(* CODESYS project proyectoFinal.project

Project tree, tasks and I/O mapping:
  Device : CODESYS Control Win V3, 3S - Smart Software Solutions GmbH, version 3.5.12.60
    application Application
      libraries: Standard, * (System)
      task MainTask (cyclic, interval t#20ms, priority 1) calls PLC_PRG
      task VISU_TASK (cyclic, interval 100 ms, priority 31) calls VisuElems.Visu_Prg
      program PLC_PRG [LD]
      visualisation Visualization
      function block LEVELMETER [LD]
      function block LEVEL_SENSORS [LD]
      function block TANK_CONTROLER [LD]
      function block LIGHTHING [LD]
      function block TIMER [LD]
      function block STATES_MACHINE [LD]
      function block TEMPERATURE_ANALOG [LD]
      function block ANALOG_TEMPERATURE [LD]
      function block TEMPERATURE_CONTROLER [LD]
      program HEATING [LD]
  text list GlobalTextList
*)

// Device/Application/PLC_PRG
	PROGRAM PLC_PRG
VAR RETAIN
	start: BOOL;
	t: TIME;
	sweet_selected: BOOL;
	acid_selected: BOOL;
	bitter_selected: BOOL;
	state_filling_mixture: BOOL;
	state_filling_solids: BOOL;
	state_sweet: BOOL;
	state_acid: BOOL;
	state_bitter: BOOL;
	state_ending: BOOL;
	state_emptying: BOOL;
	state_emergency: BOOL;
	count:BOOL;
	level: REAL;
	state_ready: BOOL;
END_VAR
VAR
	emergency_lamp: BOOL;
	speed: REAL;
	sensor_lvl_110: BOOL;
	sensed_level: REAL;
	start_button: BOOL;
	sweet_button: BOOL;
	acid_button: BOOL;
	bitter_button: BOOL;
	stop_button: BOOL;
	sensor_lvl_0: BOOL;
	sensor_lvl_60: BOOL;
	sensor_lvl_100: BOOL;
	empty_button: BOOL;
	filling_mixture_lamp: BOOL;
	filling_solids_lamp: BOOL;
	in_process_lamp: BOOL;
	sweet_selected_lamp: BOOL;
	acid_selected_lamp: BOOL;
	bitter_selected_lamp: BOOL;
	ending_lamp: BOOL;
	emptying_lamp: BOOL;
	ready_lamp: BOOL;
	reset: BOOL;
	TIMER_0: TIMER;
	STATES_MACHINE_0: STATES_MACHINE;
	LEVELMETER_0: LEVELMETER;
	LEVEL_SENSORS_0: LEVEL_SENSORS;
	TANK_CONTROLER_0: TANK_CONTROLER;
	mixer_lamp: BOOL;
	mixture_valve: BOOL;
	solids_band: BOOL;
	LIGHTHING_0: LIGHTHING;
	lighthing_lamp: BOOL;
	color: DWORD;
	wave_length: INT;
	TEMPERATURE_METER_0: TEMPERATURE_ANALOG;
	sensor_analog: REAL;
	temp: REAL:=20;
	ANALOG_TEMPERATURE_0: ANALOG_TEMPERATURE;
	sensed_temperature: REAL;
	TEMP_CONTROLER_0: TEMPERATURE_CONTROLER;
	heat: BOOL;
	empty_valve: INT;
	empty_valve_lamp: BOOL;
END_VAR
VAR // added by the converter: edge detectors and wires of the graphical bodies
    _w1 : BOOL;
END_VAR

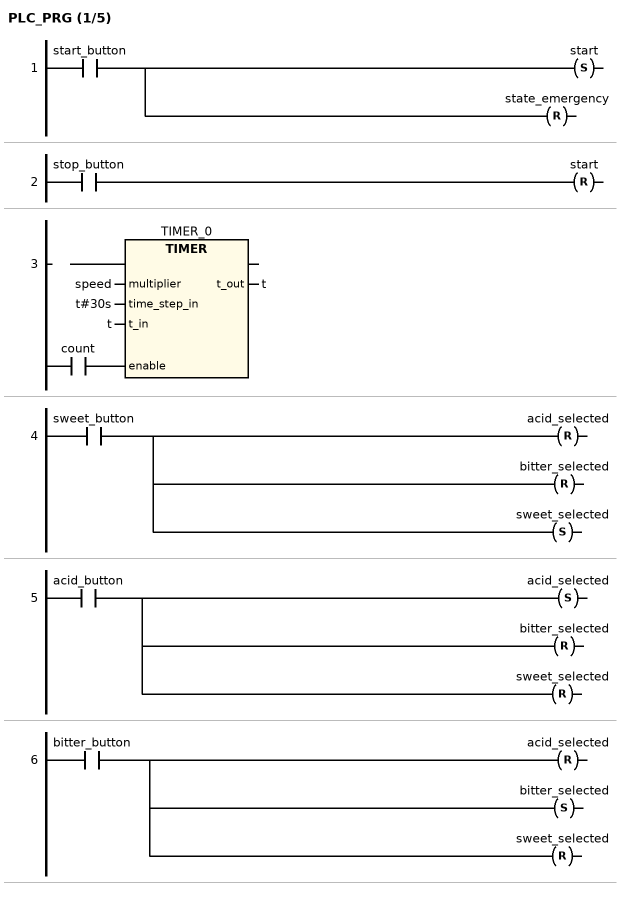
// NETWORK 1
start S= start_button;
state_emergency R= start_button;

// NETWORK 2
start R= stop_button;

// NETWORK 3
TIMER_0(multiplier := speed, time_step_in := t#30s, t_in := t, enable := count, t_out => t); // TIMER

// NETWORK 4
acid_selected R= sweet_button;
bitter_selected R= sweet_button;
sweet_selected S= sweet_button;

// NETWORK 5
acid_selected S= acid_button;
bitter_selected R= acid_button;
sweet_selected R= acid_button;

// NETWORK 6
acid_selected R= bitter_button;
bitter_selected S= bitter_button;
sweet_selected R= bitter_button;

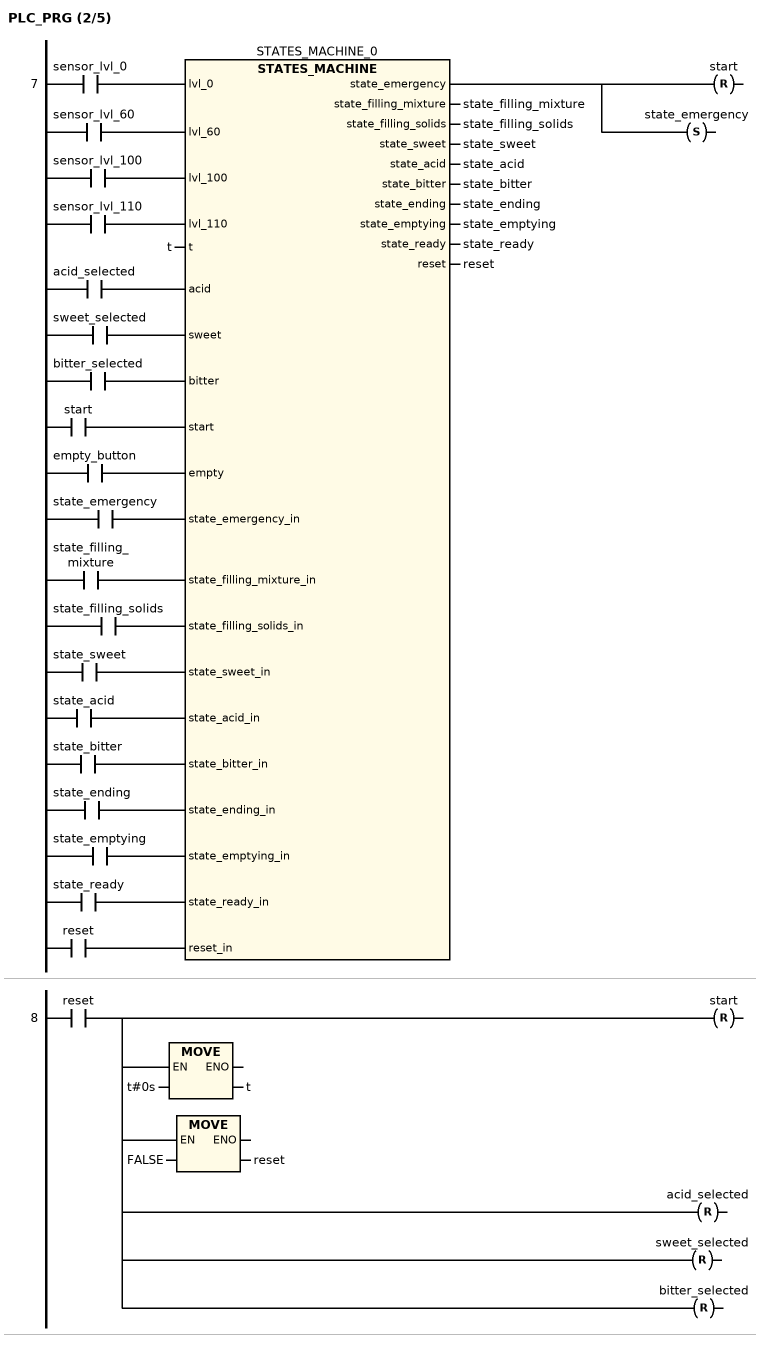
// NETWORK 7
STATES_MACHINE_0(
    lvl_0 := sensor_lvl_0,
    lvl_60 := sensor_lvl_60,
    lvl_100 := sensor_lvl_100,
    lvl_110 := sensor_lvl_110,
    t := t,
    acid := acid_selected,
    sweet := sweet_selected,
    bitter := bitter_selected,
    start := start,
    empty := empty_button,
    state_emergency_in := state_emergency,
    state_filling_mixture_in := state_filling_mixture,
    state_filling_solids_in := state_filling_solids,
    state_sweet_in := state_sweet,
    state_acid_in := state_acid,
    state_bitter_in := state_bitter,
    state_ending_in := state_ending,
    state_emptying_in := state_emptying,
    state_ready_in := state_ready,
    reset_in := reset,
    state_filling_mixture => state_filling_mixture,
    state_filling_solids => state_filling_solids,
    state_sweet => state_sweet,
    state_acid => state_acid,
    state_bitter => state_bitter,
    state_ending => state_ending,
    state_emptying => state_emptying,
    state_ready => state_ready,
    reset => reset); // STATES_MACHINE
start R= STATES_MACHINE_0.state_emergency;
state_emergency S= STATES_MACHINE_0.state_emergency;

// NETWORK 8
_w1 := reset;
start R= _w1;
IF _w1 THEN t := t#0s; END_IF
IF _w1 THEN reset := FALSE; END_IF
acid_selected R= _w1;
sweet_selected R= _w1;
bitter_selected R= _w1;

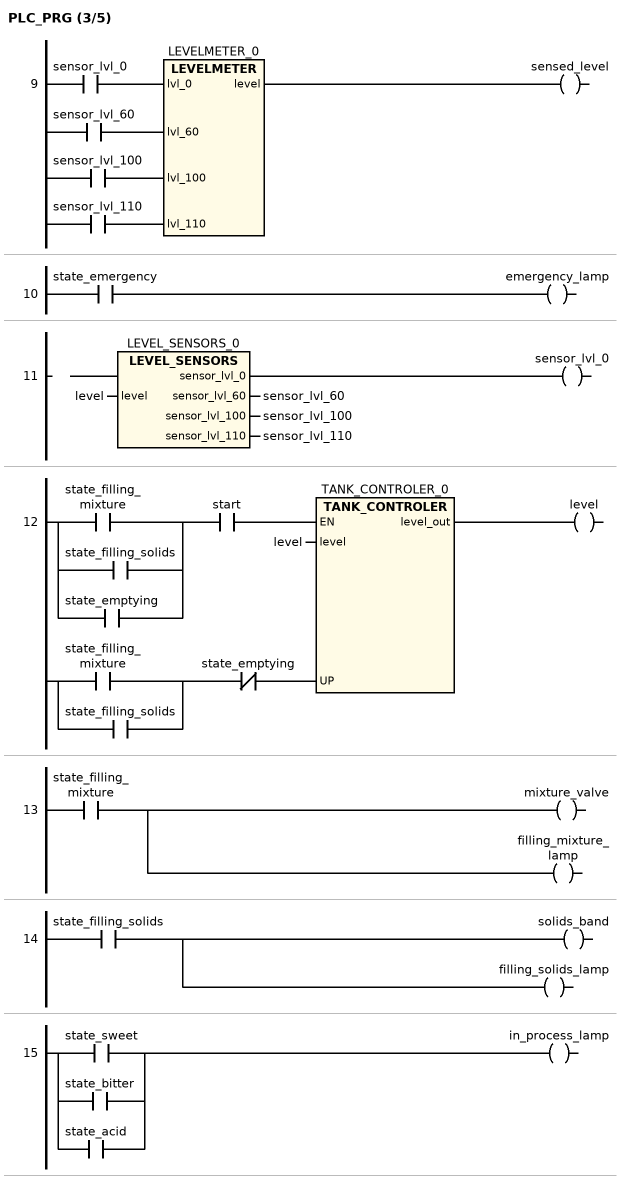
// NETWORK 9
LEVELMETER_0(
    lvl_0 := sensor_lvl_0,
    lvl_60 := sensor_lvl_60,
    lvl_100 := sensor_lvl_100,
    lvl_110 := sensor_lvl_110); // LEVELMETER
sensed_level := LEVELMETER_0.level;

// NETWORK 10
emergency_lamp := state_emergency;

// NETWORK 11
LEVEL_SENSORS_0(
    level := level,
    sensor_lvl_60 => sensor_lvl_60,
    sensor_lvl_100 => sensor_lvl_100,
    sensor_lvl_110 => sensor_lvl_110); // LEVEL_SENSORS
sensor_lvl_0 := LEVEL_SENSORS_0.sensor_lvl_0;

// NETWORK 12
TANK_CONTROLER_0(
    EN := (state_filling_mixture OR state_filling_solids OR state_emptying) AND start,
    level := level,
    UP := (state_filling_mixture OR state_filling_solids) AND NOT state_emptying); // TANK_CONTROLER
level := TANK_CONTROLER_0.level_out;

// NETWORK 13
mixture_valve := state_filling_mixture;
filling_mixture_lamp := state_filling_mixture;

// NETWORK 14
solids_band := state_filling_solids;
filling_solids_lamp := state_filling_solids;

// NETWORK 15
in_process_lamp := state_sweet OR state_bitter OR state_acid;

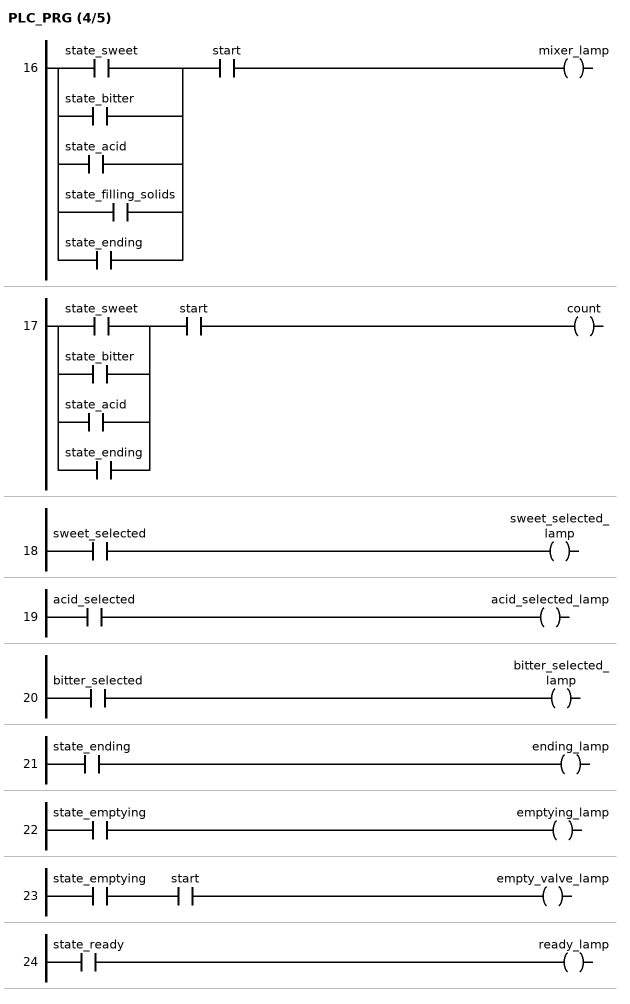
// NETWORK 16
mixer_lamp := (state_sweet OR state_bitter OR state_acid OR state_filling_solids OR state_ending) AND start;

// NETWORK 17
count := (state_sweet OR state_bitter OR state_acid OR state_ending) AND start;

// NETWORK 18
sweet_selected_lamp := sweet_selected;

// NETWORK 19
acid_selected_lamp := acid_selected;

// NETWORK 20
bitter_selected_lamp := bitter_selected;

// NETWORK 21
ending_lamp := state_ending;

// NETWORK 22
emptying_lamp := state_emptying;

// NETWORK 23
empty_valve_lamp := state_emptying AND start;

// NETWORK 24
ready_lamp := state_ready;

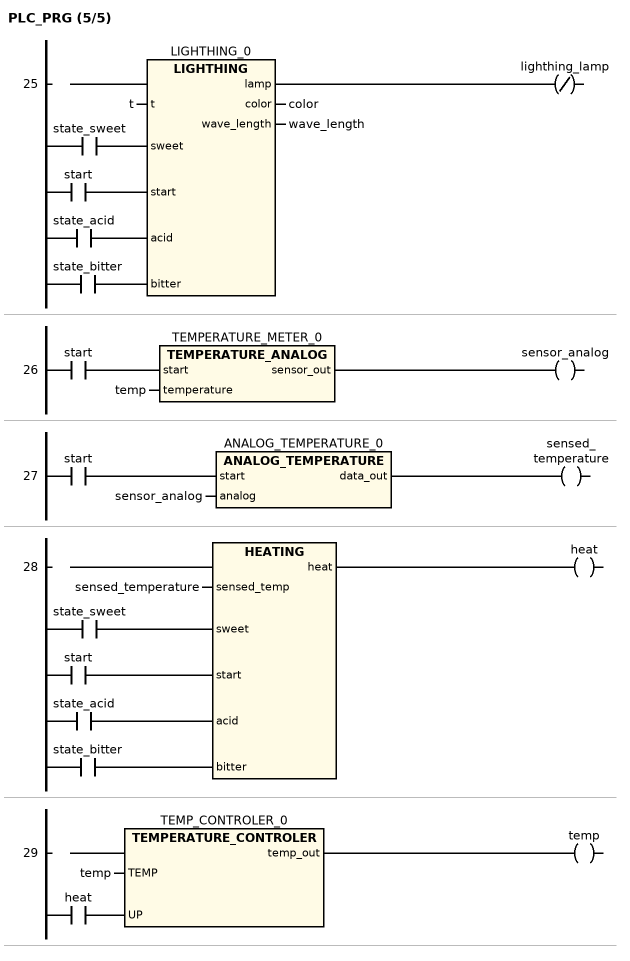
// NETWORK 25
LIGHTHING_0(
    t := t,
    sweet := state_sweet,
    start := start,
    acid := state_acid,
    bitter := state_bitter,
    color => color,
    wave_length => wave_length); // LIGHTHING
lighthing_lamp := NOT LIGHTHING_0.lamp;

// NETWORK 26
TEMPERATURE_METER_0(start := start, temperature := temp); // TEMPERATURE_ANALOG
sensor_analog := TEMPERATURE_METER_0.sensor_out;

// NETWORK 27
ANALOG_TEMPERATURE_0(start := start, analog := sensor_analog); // ANALOG_TEMPERATURE
sensed_temperature := ANALOG_TEMPERATURE_0.data_out;

// NETWORK 28
HEATING(sensed_temp := sensed_temperature, sweet := state_sweet, start := start, acid := state_acid, bitter := state_bitter);
heat := HEATING.heat;

// NETWORK 29
TEMP_CONTROLER_0(TEMP := temp, UP := heat); // TEMPERATURE_CONTROLER
temp := TEMP_CONTROLER_0.temp_out;

END_PROGRAM

// Device/Application/TIMER
FUNCTION_BLOCK TIMER
VAR_INPUT
	multiplier: REAL:=1;
	time_step_in: TIME;
	t_in: TIME;
	enable: BOOL;
	reset: BOOL;
END_VAR
VAR_OUTPUT
	t_out:TIME;
END_VAR
VAR
	TOF_0: TOF;
	time_step_real: REAL;
	time_step_in_real: REAL;
	time_step: TIME;
END_VAR

VAR_TEMP
	t: TIME;
END_VAR

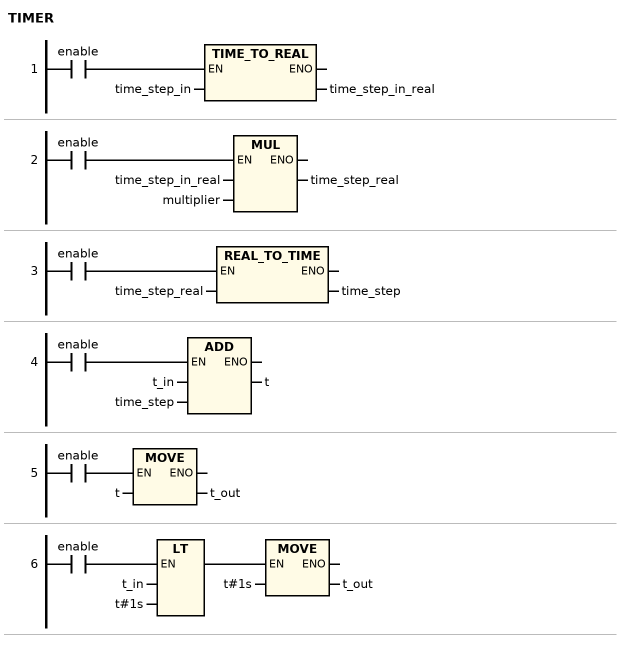
// NETWORK 1
IF enable THEN time_step_in_real := TIME_TO_REAL(time_step_in); END_IF

// NETWORK 2
IF enable THEN time_step_real := time_step_in_real * multiplier; END_IF

// NETWORK 3
IF enable THEN time_step := REAL_TO_TIME(time_step_real); END_IF

// NETWORK 4
IF enable THEN t := t_in + time_step; END_IF

// NETWORK 5
IF enable THEN t_out := t; END_IF

// NETWORK 6
IF enable AND t_in < t#1s THEN t_out := t#1s; END_IF

END_FUNCTION_BLOCK

// Device/Application/STATES_MACHINE
FUNCTION_BLOCK STATES_MACHINE
VAR_INPUT
	lvl_0 :BOOL;
	lvl_60 :BOOL;
	lvl_100 :BOOL;
	lvl_110 :BOOL;
	t :TIME;
	acid: BOOL;
	sweet: BOOL;
	bitter: BOOL;
	start: BOOL;
	empty: BOOL;
	state_emergency_in: BOOL;
	state_filling_mixture_in:BOOL;
	state_filling_solids_in:BOOL;
	state_sweet_in:BOOL;
	state_acid_in:BOOL;
	state_bitter_in:BOOL;
	state_ending_in:BOOL;
	state_emptying_in:BOOL;
	state_ready_in: BOOL;
	reset_in: BOOL;
END_VAR
VAR_OUTPUT
	state_emergency: BOOL;
	state_filling_mixture:BOOL;
	state_filling_solids:BOOL;
	state_sweet:BOOL;
	state_acid:BOOL;
	state_bitter:BOOL;
	state_ending:BOOL;
	state_emptying:BOOL;
	state_ready: BOOL;
	reset: BOOL;
END_VAR
VAR
	emergency: BOOL;
END_VAR
VAR // added by the converter: edge detectors and wires of the graphical bodies
    _w1, _w2, _w3, _w4, _w5, _w6, _w7, _w8, _w9, _w10 : BOOL;
END_VAR

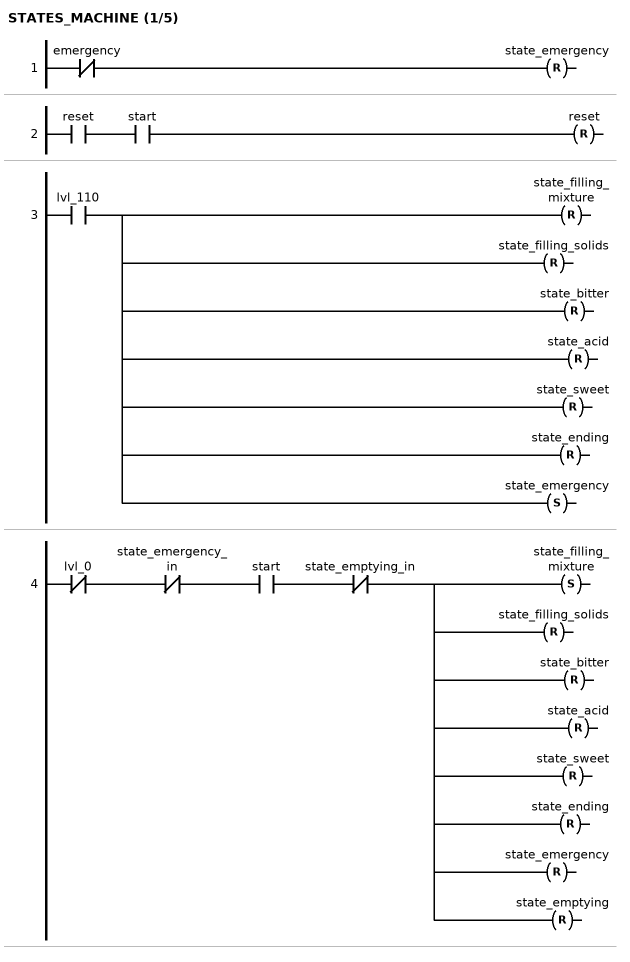
// NETWORK 1
state_emergency R= NOT emergency;

// NETWORK 2
reset R= reset AND start;

// NETWORK 3
state_filling_mixture R= lvl_110;
state_filling_solids R= lvl_110;
state_bitter R= lvl_110;
state_acid R= lvl_110;
state_sweet R= lvl_110;
state_ending R= lvl_110;
state_emergency S= lvl_110;

// NETWORK 4
_w1 := NOT lvl_0 AND NOT state_emergency_in AND start AND NOT state_emptying_in;
state_filling_mixture S= _w1;
state_filling_solids R= _w1;
state_bitter R= _w1;
state_acid R= _w1;
state_sweet R= _w1;
state_ending R= _w1;
state_emergency R= _w1;
state_emptying R= _w1;

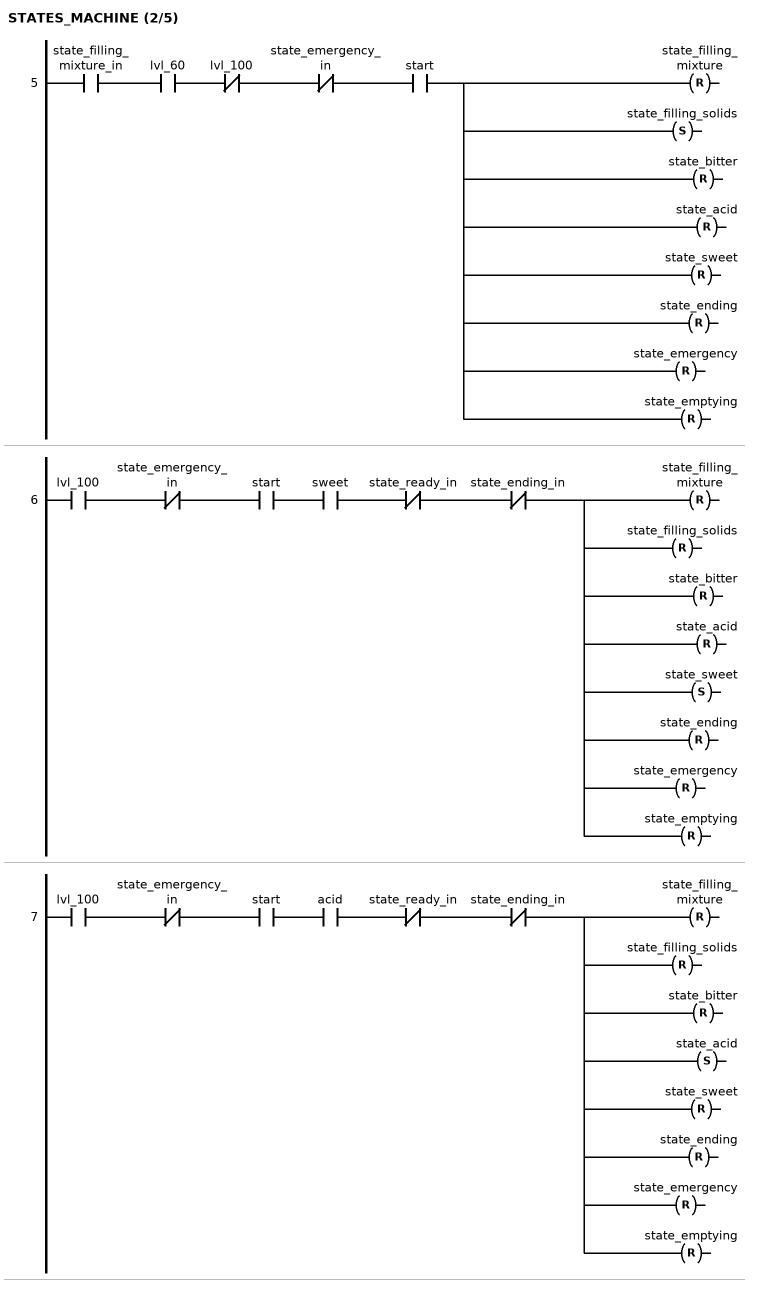
// NETWORK 5
_w2 := state_filling_mixture_in AND lvl_60 AND NOT lvl_100 AND NOT state_emergency_in AND start;
state_filling_mixture R= _w2;
state_filling_solids S= _w2;
state_bitter R= _w2;
state_acid R= _w2;
state_sweet R= _w2;
state_ending R= _w2;
state_emergency R= _w2;
state_emptying R= _w2;

// NETWORK 6
_w3 := lvl_100 AND NOT state_emergency_in AND start AND sweet AND NOT state_ready_in AND NOT state_ending_in;
state_filling_mixture R= _w3;
state_filling_solids R= _w3;
state_bitter R= _w3;
state_acid R= _w3;
state_sweet S= _w3;
state_ending R= _w3;
state_emergency R= _w3;
state_emptying R= _w3;

// NETWORK 7
_w4 := lvl_100 AND NOT state_emergency_in AND start AND acid AND NOT state_ready_in AND NOT state_ending_in;
state_filling_mixture R= _w4;
state_filling_solids R= _w4;
state_bitter R= _w4;
state_acid S= _w4;
state_sweet R= _w4;
state_ending R= _w4;
state_emergency R= _w4;
state_emptying R= _w4;

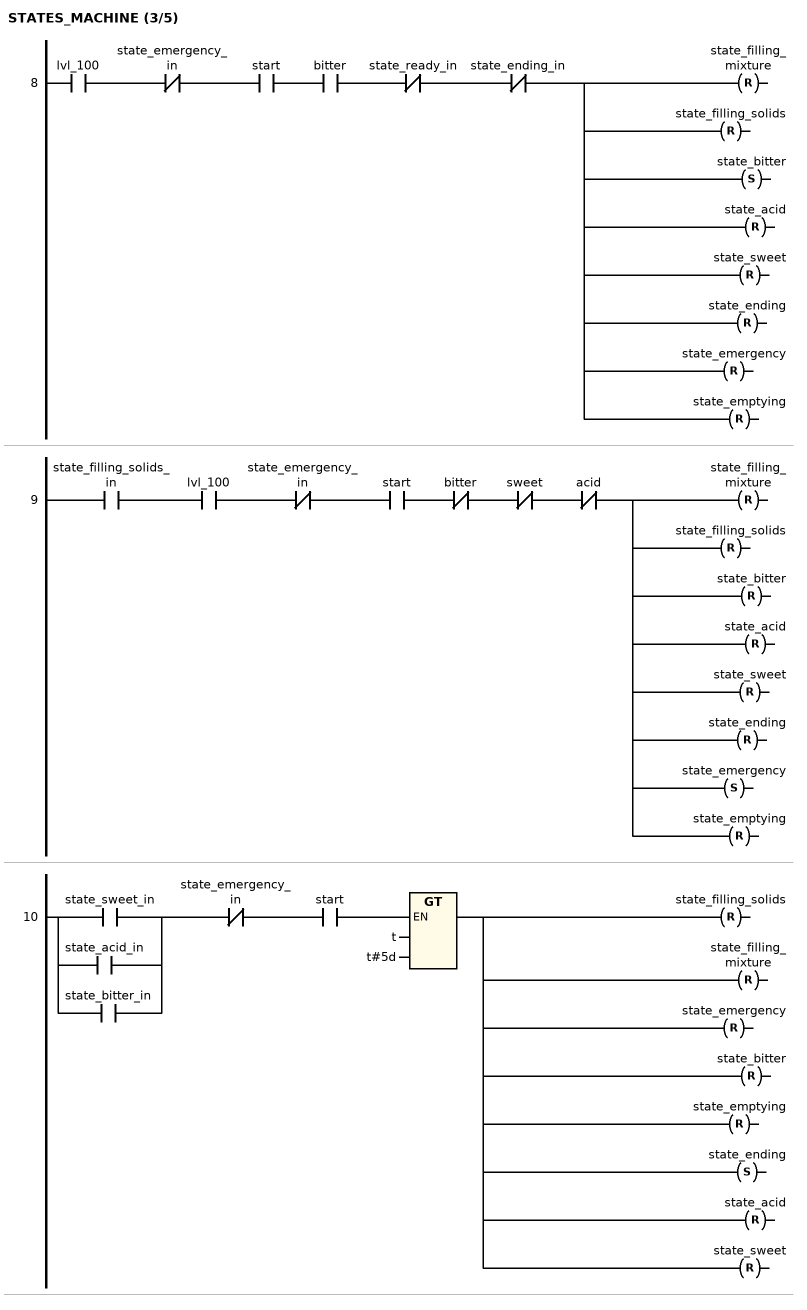
// NETWORK 8
_w5 := lvl_100 AND NOT state_emergency_in AND start AND bitter AND NOT state_ready_in AND NOT state_ending_in;
state_filling_mixture R= _w5;
state_filling_solids R= _w5;
state_bitter S= _w5;
state_acid R= _w5;
state_sweet R= _w5;
state_ending R= _w5;
state_emergency R= _w5;
state_emptying R= _w5;

// NETWORK 9
_w6 := state_filling_solids_in AND lvl_100 AND NOT state_emergency_in AND start AND NOT bitter AND NOT sweet AND NOT acid;
state_filling_mixture R= _w6;
state_filling_solids R= _w6;
state_bitter R= _w6;
state_acid R= _w6;
state_sweet R= _w6;
state_ending R= _w6;
state_emergency S= _w6;
state_emptying R= _w6;

// NETWORK 10
_w7 := (state_sweet_in OR state_acid_in OR state_bitter_in) AND NOT state_emergency_in AND start AND t > t#5d;
state_filling_solids R= _w7;
state_filling_mixture R= _w7;
state_emergency R= _w7;
state_bitter R= _w7;
state_emptying R= _w7;
state_ending S= _w7;
state_acid R= _w7;
state_sweet R= _w7;

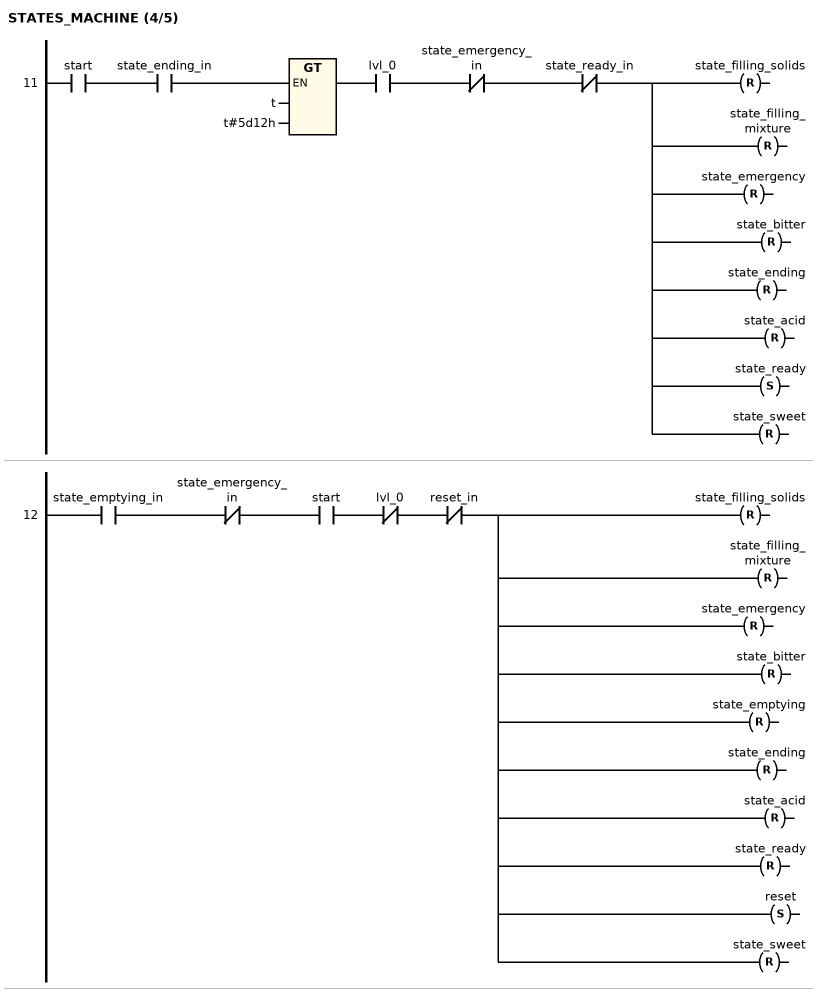
// NETWORK 11
_w8 := (start AND state_ending_in AND t > t#5d12h) AND lvl_0 AND NOT state_emergency_in AND NOT state_ready_in;
state_filling_solids R= _w8;
state_filling_mixture R= _w8;
state_emergency R= _w8;
state_bitter R= _w8;
state_ending R= _w8;
state_acid R= _w8;
state_ready S= _w8;
state_sweet R= _w8;

// NETWORK 12
_w9 := state_emptying_in AND NOT state_emergency_in AND start AND NOT lvl_0 AND NOT reset_in;
state_filling_solids R= _w9;
state_filling_mixture R= _w9;
state_emergency R= _w9;
state_bitter R= _w9;
state_emptying R= _w9;
state_ending R= _w9;
state_acid R= _w9;
state_ready R= _w9;
reset S= _w9;
state_sweet R= _w9;

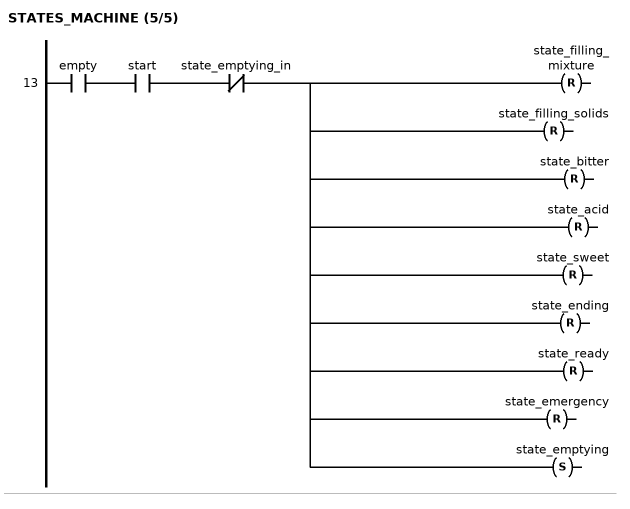
// NETWORK 13
_w10 := empty AND start AND NOT state_emptying_in;
state_filling_mixture R= _w10;
state_filling_solids R= _w10;
state_bitter R= _w10;
state_acid R= _w10;
state_sweet R= _w10;
state_ending R= _w10;
state_ready R= _w10;
state_emergency R= _w10;
state_emptying S= _w10;

END_FUNCTION_BLOCK

// Device/Application/LEVELMETER
FUNCTION_BLOCK LEVELMETER
VAR_INPUT
	lvl_0: BOOL;
	lvl_60: BOOL;
	lvl_100: BOOL;
	lvl_110: BOOL;
END_VAR
VAR_OUTPUT
	level: REAL;
END_VAR
VAR
	lvl_1: BOOL;
END_VAR

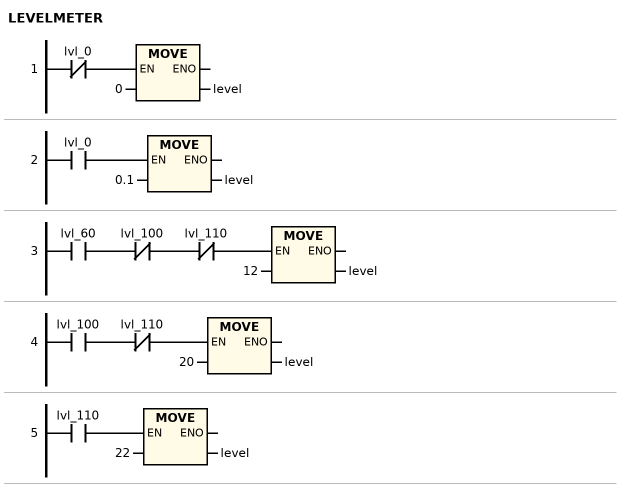
// NETWORK 1
IF NOT lvl_0 THEN level := 0; END_IF

// NETWORK 2
IF lvl_0 THEN level := 0.1; END_IF

// NETWORK 3
IF lvl_60 AND NOT lvl_100 AND NOT lvl_110 THEN level := 12; END_IF

// NETWORK 4
IF lvl_100 AND NOT lvl_110 THEN level := 20; END_IF

// NETWORK 5
IF lvl_110 THEN level := 22; END_IF

END_FUNCTION_BLOCK

// Device/Application/LEVEL_SENSORS
FUNCTION_BLOCK LEVEL_SENSORS
VAR_INPUT
	level: REAL;
END_VAR
VAR_OUTPUT
	sensor_lvl_0: BOOL;
	sensor_lvl_60: BOOL;
	sensor_lvl_100: BOOL;
	sensor_lvl_110: BOOL;
END_VAR
VAR // added by the converter: edge detectors and wires of the graphical bodies
    _w1, _w2, _w3, _w4 : BOOL;
END_VAR

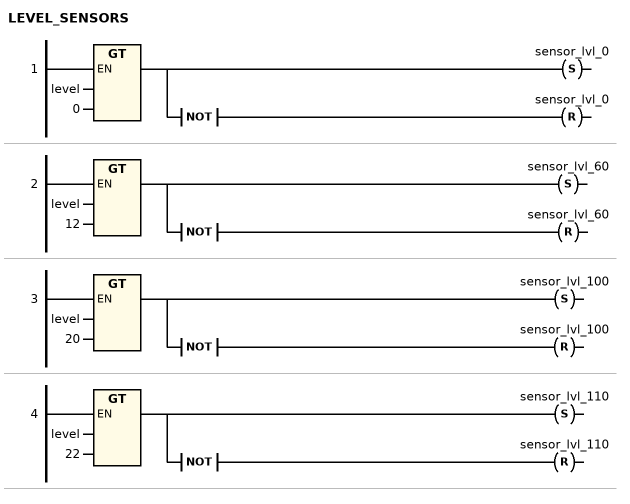
// NETWORK 1
_w1 := level > 0;
sensor_lvl_0 S= _w1;
sensor_lvl_0 R= NOT _w1;

// NETWORK 2
_w2 := level > 12;
sensor_lvl_60 S= _w2;
sensor_lvl_60 R= NOT _w2;

// NETWORK 3
_w3 := level > 20;
sensor_lvl_100 S= _w3;
sensor_lvl_100 R= NOT _w3;

// NETWORK 4
_w4 := level > 22;
sensor_lvl_110 S= _w4;
sensor_lvl_110 R= NOT _w4;

END_FUNCTION_BLOCK

// Device/Application/TANK_CONTROLER
FUNCTION_BLOCK TANK_CONTROLER
VAR_INPUT
	EN: BOOL;
	level: REAL;
	UP: BOOL;
END_VAR
VAR_OUTPUT
	level_out: REAL;
END_VAR

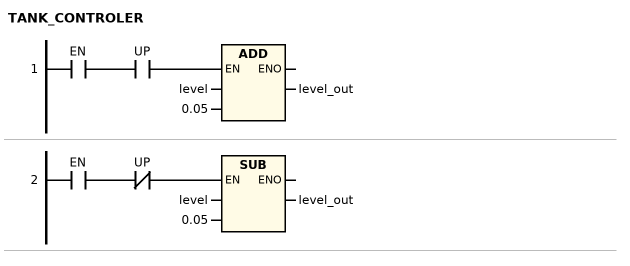
// NETWORK 1
IF EN AND UP THEN level_out := level + 0.05; END_IF

// NETWORK 2
IF EN AND NOT UP THEN level_out := level - 0.05; END_IF

END_FUNCTION_BLOCK

// Device/Application/LIGHTHING
FUNCTION_BLOCK LIGHTHING
VAR_INPUT
	t: TIME;
	sweet: BOOL;
	start: BOOL;
	acid: BOOL;
	bitter: BOOL;
END_VAR
VAR_OUTPUT
	lamp: BOOL;
	color: DWORD;
	wave_length: INT;
END_VAR
VAR
	t_int: UDINT;
	day_int: UDINT;
	module: UDINT;
	module_time: TIME;
	lamp_sweet: BOOL;
	lamp_acid: BOOL;
	lamp_bitter: BOOL;
END_VAR
VAR // added by the converter: edge detectors and wires of the graphical bodies
    _w1, _w2, _w3 : BOOL;
END_VAR

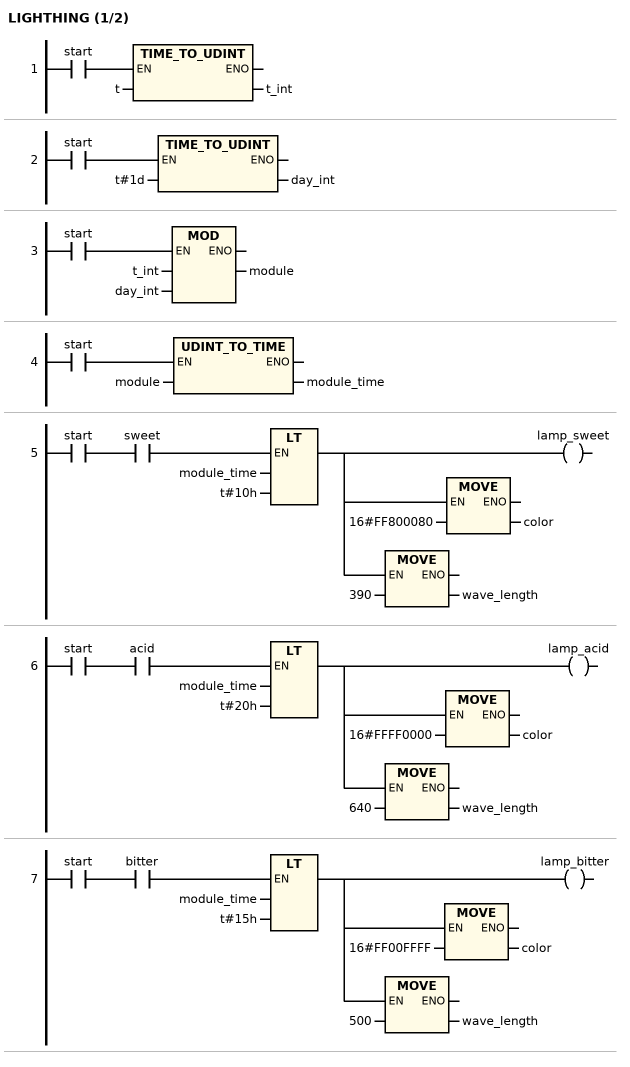
// NETWORK 1
IF start THEN t_int := TIME_TO_UDINT(t); END_IF

// NETWORK 2
IF start THEN day_int := TIME_TO_UDINT(t#1d); END_IF

// NETWORK 3
IF start THEN module := t_int MOD day_int; END_IF

// NETWORK 4
IF start THEN module_time := UDINT_TO_TIME(module); END_IF

// NETWORK 5
_w1 := start AND sweet AND module_time < t#10h;
lamp_sweet := _w1;
IF _w1 THEN color := 16#FF800080; END_IF
IF _w1 THEN wave_length := 390; END_IF

// NETWORK 6
_w2 := start AND acid AND module_time < t#20h;
lamp_acid := _w2;
IF _w2 THEN color := 16#FFFF0000; END_IF
IF _w2 THEN wave_length := 640; END_IF

// NETWORK 7
_w3 := start AND bitter AND module_time < t#15h;
lamp_bitter := _w3;
IF _w3 THEN color := 16#FF00FFFF; END_IF
IF _w3 THEN wave_length := 500; END_IF

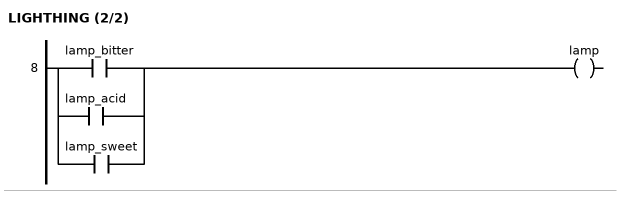
// NETWORK 8
lamp := lamp_bitter OR lamp_acid OR lamp_sweet;

END_FUNCTION_BLOCK

// Device/Application/TEMPERATURE_ANALOG
FUNCTION_BLOCK TEMPERATURE_ANALOG
VAR_INPUT
	start: BOOL;
	temperature: REAL;
END_VAR
VAR_OUTPUT
		sensor_out: REAL;
END_VAR
VAR
	num: REAL;
	den: REAL;
	A: REAL;
	mult: REAL;
	sub1: REAL;
END_VAR

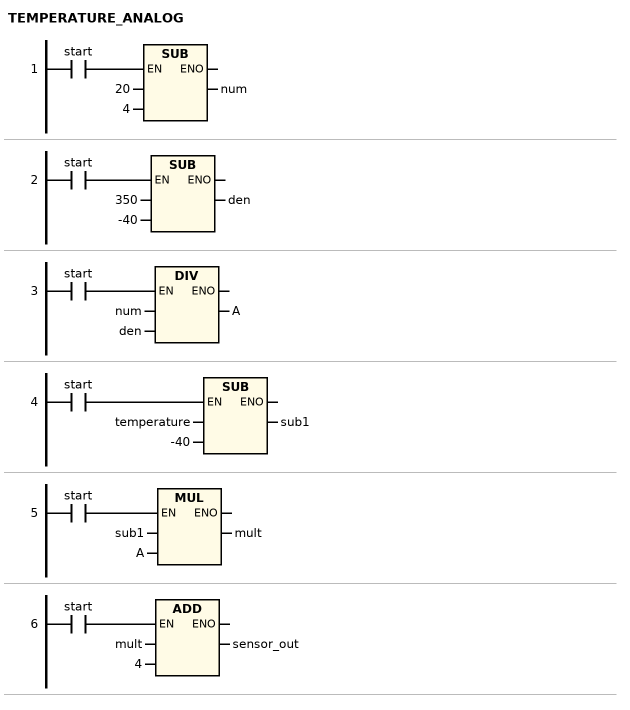
// NETWORK 1
IF start THEN num := 20 - 4; END_IF

// NETWORK 2
IF start THEN den := 350 - -40; END_IF

// NETWORK 3
IF start THEN A := num / den; END_IF

// NETWORK 4
IF start THEN sub1 := temperature - -40; END_IF

// NETWORK 5
IF start THEN mult := sub1 * A; END_IF

// NETWORK 6
IF start THEN sensor_out := mult + 4; END_IF

END_FUNCTION_BLOCK

// Device/Application/ANALOG_TEMPERATURE
FUNCTION_BLOCK ANALOG_TEMPERATURE
VAR_INPUT
	start: BOOL;
	analog: REAL;
END_VAR
VAR_OUTPUT
	data_out: REAL;
END_VAR
VAR
	num: REAL;
	den: REAL;
	A: REAL;
	mult: REAL;
	sub1: REAL;
END_VAR

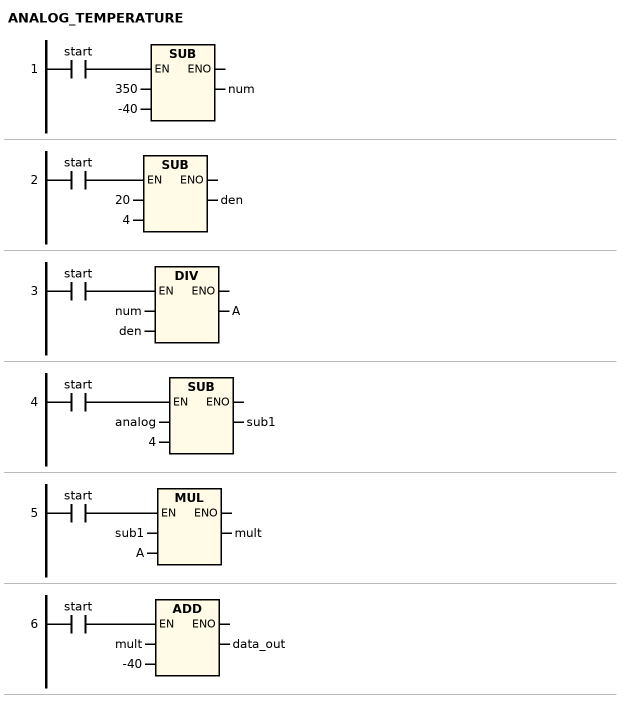
// NETWORK 1
IF start THEN num := 350 - -40; END_IF

// NETWORK 2
IF start THEN den := 20 - 4; END_IF

// NETWORK 3
IF start THEN A := num / den; END_IF

// NETWORK 4
IF start THEN sub1 := analog - 4; END_IF

// NETWORK 5
IF start THEN mult := sub1 * A; END_IF

// NETWORK 6
IF start THEN data_out := mult + -40; END_IF

END_FUNCTION_BLOCK

// Device/Application/HEATING
PROGRAM HEATING
VAR_INPUT
	sensed_temp:REAL;
	sweet: BOOL;
	start: BOOL;
	acid: BOOL;
	bitter: BOOL;
END_VAR
VAR_OUTPUT
 heat: BOOL;
END_VAR
VAR
END_VAR

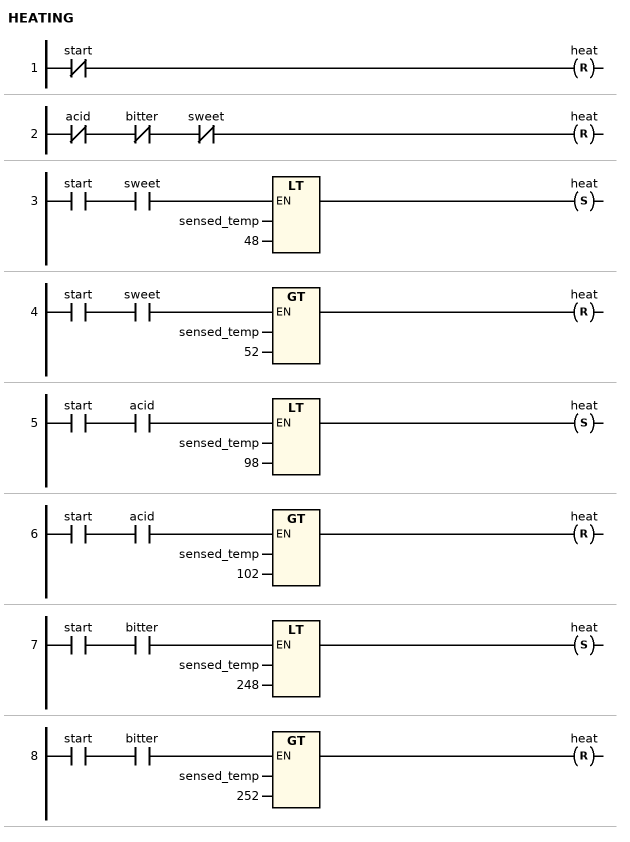
// NETWORK 1
heat R= NOT start;

// NETWORK 2
heat R= NOT acid AND NOT bitter AND NOT sweet;

// NETWORK 3
heat S= start AND sweet AND sensed_temp < 48;

// NETWORK 4
heat R= start AND sweet AND sensed_temp > 52;

// NETWORK 5
heat S= start AND acid AND sensed_temp < 98;

// NETWORK 6
heat R= start AND acid AND sensed_temp > 102;

// NETWORK 7
heat S= start AND bitter AND sensed_temp < 248;

// NETWORK 8
heat R= start AND bitter AND sensed_temp > 252;

END_PROGRAM

// Device/Application/TEMPERATURE_CONTROLER
FUNCTION_BLOCK TEMPERATURE_CONTROLER
VAR_INPUT
	TEMP: REAL;
	UP: BOOL;
END_VAR
VAR_OUTPUT
	temp_out: REAL;
END_VAR

VAR
	lowest: BOOL;
	highest: BOOL;
END_VAR

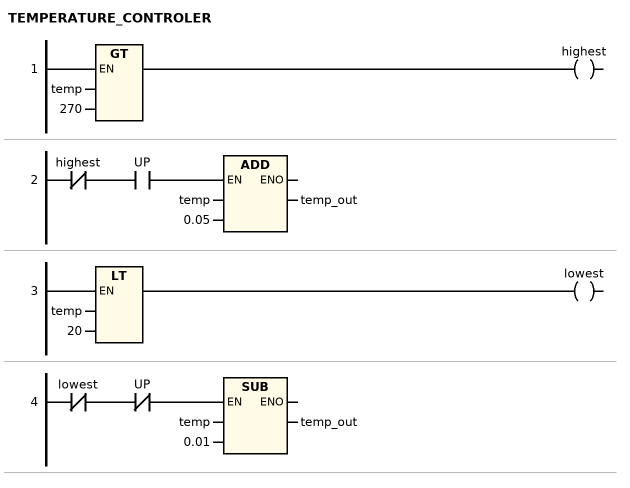
// NETWORK 1
highest := temp > 270;

// NETWORK 2
IF NOT highest AND UP THEN temp_out := temp + 0.05; END_IF

// NETWORK 3
lowest := temp < 20;

// NETWORK 4
IF NOT lowest AND NOT UP THEN temp_out := temp - 0.01; END_IF

END_FUNCTION_BLOCK

// Device/Application/Visualization
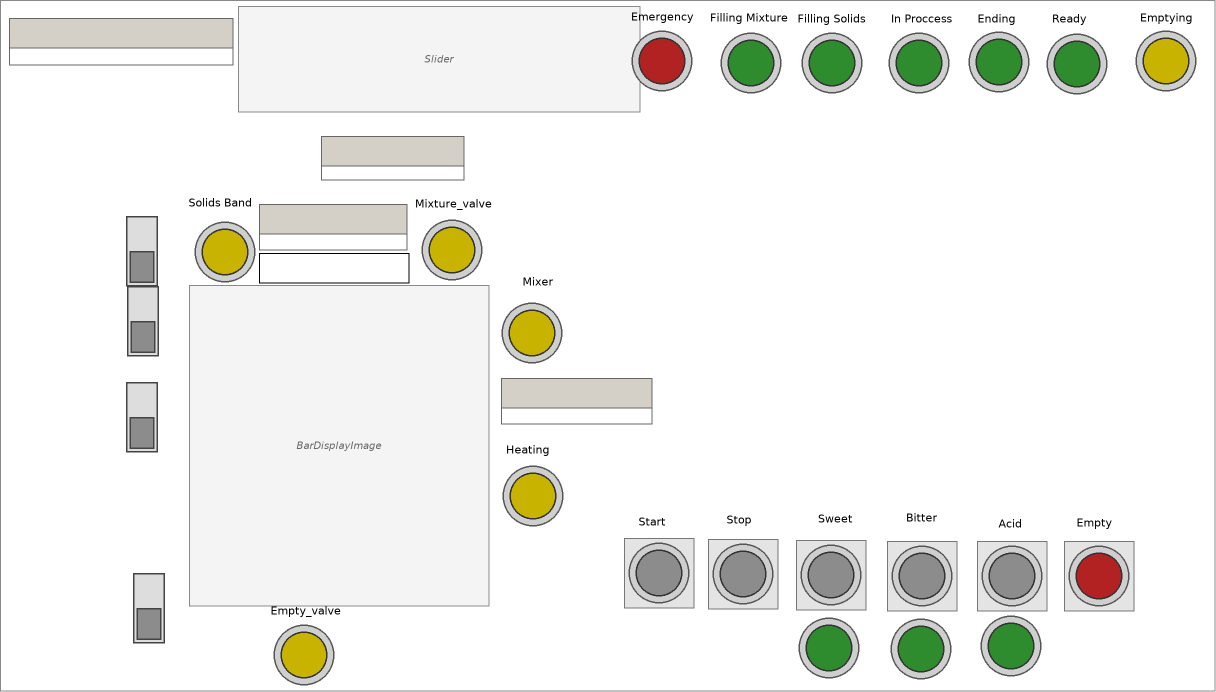
VISUALIZATION Visualization  // 1216x692
    Table (9,18 224x47), data array: PLC_PRG.t
        p3854506369: PLC_PRG.t
        p2232123230: Time
    Slider (238,6 402x106), variable: PLC_PRG.speed, scale 0..10
    Label (621,507 62x30), "Start"
    Table (321,136 143x44), data array: PLC_PRG.speed
        p3854506369: PLC_PRG.speed
        p2232123230: Speed
    PushSwitch (624,538 70x70), variable: PLC_PRG.start_button, behaviour: TAP, style: Switch-PushSwitch-Gray
    PushSwitch (708,539 70x70), variable: PLC_PRG.stop_button, behaviour: TAP, style: Switch-PushSwitch-Gray
    Label (708,505 62x30), "Stop"
    Lamp1 (627,26 70x70), variable: PLC_PRG.state_emergency, style: Lamp-Lamp1-Red
    Label (615,2 95x30), "Emergency"
    DipSwitch (107,216 70x70), variable: PLC_PRG.sensor_lvl_110, behaviour: TOGGLE, style: Switch-DipSwitch-Gray
    DipSwitch (108,286 70x70), variable: PLC_PRG.sensor_lvl_100, behaviour: TOGGLE, style: Switch-DipSwitch-Gray
    DipSwitch (107,382 70x70), variable: PLC_PRG.sensor_lvl_60, behaviour: TOGGLE, style: Switch-DipSwitch-Gray
    DipSwitch (114,573 70x70), variable: PLC_PRG.sensor_lvl_0, behaviour: TOGGLE, style: Switch-DipSwitch-Gray
    BarDisplayImage (189,285 300x321), value: PLC_PRG.sensed_level, style: BarDisplayImage-Gray, scale format: %.1f, scale 0..20
    Lamp1 (716,28 70x70), variable: PLC_PRG.filling_mixture_lamp, style: Lamp-Lamp1-Green
    Label (1119,3 95x30), "Emptying"
    Label (949,4 95x30), "Ending"
    Label (788,504 95x30), "Sweet"
    Label (874,4 95x30), "In Proccess"
    Label (784,4 95x30), "Filling Solids"
    Label (696,3 106x30), "Filling Mixture"
    Lamp1 (797,28 70x70), variable: PLC_PRG.filling_solids_lamp, style: Lamp-Lamp1-Green
    Lamp1 (884,28 70x70), variable: PLC_PRG.in_process_lamp, style: Lamp-Lamp1-Green
    Label (874,503 95x30), "Bitter"
    Label (963,509 95x30), "Acid"
    PushSwitch (796,540 70x70), variable: PLC_PRG.sweet_button, behaviour: TAP, style: Switch-PushSwitch-Gray
    PushSwitch (887,541 70x70), variable: PLC_PRG.bitter_button, behaviour: TAP, style: Switch-PushSwitch-Gray
    PushSwitch (977,541 70x70), variable: PLC_PRG.acid_button, behaviour: TAP, style: Switch-PushSwitch-Gray
    Lamp1 (794,613 70x70), variable: PLC_PRG.sweet_selected_lamp, style: Lamp-Lamp1-Green
    Lamp1 (886,614 70x70), variable: PLC_PRG.bitter_selected_lamp, style: Lamp-Lamp1-Green
    Lamp1 (976,611 70x70), variable: PLC_PRG.acid_selected_lamp, style: Lamp-Lamp1-Green
    Lamp1 (964,27 70x70), variable: PLC_PRG.ending_lamp, style: Lamp-Lamp1-Green
    Lamp1 (1131,26 70x70), variable: PLC_PRG.emptying_lamp, style: Lamp-Lamp1-Yellow
    Lamp1 (1042,29 70x70), variable: PLC_PRG.ready_lamp, style: Lamp-Lamp1-Green
    Label (1022,4 95x30), "Ready"
    PushSwitch (1064,541 70x70), variable: PLC_PRG.empty_button, behaviour: TAP, style: Switch-PushSwitch-Red
    Label (1047,508 95x30), "Empty"
    Lamp1 (497,298 70x70), variable: PLC_PRG.mixer_lamp, style: Lamp-Lamp1-Yellow
    Label (507,267 62x30), "Mixer"
    Lamp1 (417,215 70x70), variable: PLC_PRG.mixture_valve, style: Lamp-Lamp1-Yellow
    Label (398,189 111x30), "Mixture_valve"
    Lamp1 (190,217 70x70), variable: PLC_PRG.solids_band, style: Lamp-Lamp1-Yellow
    Label (165,188 111x30), "Solids Band"
    RoundedRectangle (259,253 150x30), colour toggle: PLC_PRG.lighthing_lamp, invisible if: PLC_PRG.lighthing_lamp, colour variable: PLC_PRG.color
    Table (259,204 148x46), data array: PLC_PRG.wave_length
        p3854506369: PLC_PRG.wave_length
        p2232123230: Wave Length (nm)
    Table (501,378 151x46), data array: PLC_PRG.sensed_temperature
        p3854506369: PLC_PRG.sensed_temperature
        p2232123230: Temperature ( C°)
    Lamp1 (269,620 70x70), variable: PLC_PRG.empty_valve_lamp, style: Lamp-Lamp1-Yellow
    Label (264,596 84x30), "Empty_valve"
    Lamp1 (498,461 70x70), variable: PLC_PRG.heat, style: Lamp-Lamp1-Yellow
    Label (497,435 62x30), "Heating"
END_VISUALIZATION
